FUNCTION_BLOCK SlitPairs
VAR_INPUT
	gap		:	AXIS_REF;
	centre	:	AXIS_REF;
	blade1	:	AXIS_REF;
	blade2	:	AXIS_REF;
	bCoupled	:	BOOL;
END_VAR
VAR_OUTPUT
END_VAR
VAR
	iState	:	UINT;
	MCCamInG	:	MC_CamIn_V2;
	MCCamInC	:	MC_CamIn_V2;
	MCCamAddG	:	MC_CamAdd;	
	MCCamAddC	:	MC_CamAdd;
	
	MCCamInB1	:	MC_CamIn_V2;
	MCCamInB2	:	MC_CamIn_V2;
	MCCamAddB1	:	MC_CamAdd;
	MCCamAddB2	:	MC_CamAdd;
	
	MCCamOutB1	:	MC_CamOut;
	MCCamOutB2	:	MC_CamOut;
	MCCamOutG	:	MC_CamOut;
	MCCamOutC	:	MC_CamOut;


	MCSetPosG	:	MC_SetPosition;
	MCSetPosC	:	MC_SetPosition;
	gapVal		:	LREAL;
	centVal		:	LREAL;
	

	
	
	
END_VAR

MCCamInB1(Master:=gap, Slave:=blade1);
MCCamAddB1(Master:=centre, Slave:=blade1);
MCCamInB2(Master:=gap, Slave:=blade2);
MCCamAddB2(Master:=centre, Slave:=blade2);

MCCamInG(Master:=blade1,Slave:=gap);
MCCamAddG(Master:=blade2, Slave:=gap);
MCCamInC(Master:=blade1, Slave:=centre);
MCCamAddC(Master:=blade2, Slave:=centre);

MCCamOutB1(Slave:=blade1);
MCCamOutB2(Slave:=blade2);
MCCamOutG(Slave:=gap);
MCCamOutC(Slave:=centre);


CASE iState OF
	0:	
		IF bCoupled THEN
			iState:=1;		//blades are slaves
		ELSE
			iState:= 30;		//blades are masters
		END_IF
	
	1:	//CAM IN THE GAP
		MCCamInB1(Master:=gap,Slave:=blade1,Execute:=TRUE,CamTableID:=1);
		MCCamInB2(Master:=gap,Slave:=blade2,Execute:=TRUE,CamTableID:=2);
		iState:=2;
	2:	//WAIT FOR CAM IN
		IF MCCamInB1.InSync AND MCCamInB2.InSync THEN
			MCCamInB1(Master:=gap,Slave:=blade1, Execute:=FALSE);
			MCCamInB2(Master:=gap,Slave:=blade2, Execute:=FALSE);
			iState:=3;
		END_IF
		
	3:	//CAM IN CENTRE
		MCCamAddB1(Master:=centre,Slave:=blade1,Execute:=TRUE,CamTableID:=3);
		MCCamAddB2(Master:=centre,Slave:=blade2,Execute:=TRUE,CamTableID:=4);
		iState:=4;
	4:	//WAIT FOR CAM IN
		IF MCCamAddB1.InSync AND MCCamAddB2.InSync THEN
			MCCamAddB1(Master:=centre,Slave:=blade1, Execute:=FALSE);
			MCCamAddB2(Master:=centre,Slave:=blade2, Execute:=FALSE);
			iState:=10;
		END_IF
	
	10:	//blades are slaves, do nothing unless this setup changes
		IF NOT bCoupled THEN
			iState:=20; //This is coming from slave blades, we now want to switch to gap and centre slaves so need to cam out first
		END_IF
		
	
		
	20:	//CAM OUT THE BLADES
		MCCamOutB1(Slave:=blade1, Execute:=TRUE);
		MCCamOutB2(Slave:=blade2, Execute:=TRUE);
		iState:=21;
	21:
		IF MCCamOutB1.Done AND MCCamOutB2.Done THEN
			MCCamOutB1(Slave:=blade1, Execute:=FALSE);
			MCCamOutB2(Slave:=blade2, Execute:=FALSE);
			iState:=30;	//CAMMED OUT READY FOR CAM IN
		END_IF

		
	30:	//CAM IN THE GAP AND CENTRES
		MCCamInG(Master:=blade1, Slave:=gap, Execute:=TRUE, CamTableID:= 5);
		MCCamInC(Master:=blade1, Slave:=centre, Execute:=TRUE, CamTableID:=6);
		iState:=31;
	
	31:
		IF MCCamInG.InSync AND MCCamInC.InSync THEN
			MCCamInG(Master:=blade1, Slave:=gap, Execute:=FALSE);
			MCCamInC(Master:=blade1, Slave:=centre, Execute:=FALSE);
			iState:=32;
		END_IF
	32:	//MULTI CAM
		MCCamAddG(Master:=blade2, Slave:=gap, Execute:=TRUE, CamTableID:=7);
		MCCamAddC(Master:=blade2, Slave:=centre, Execute:=TRUE, CamTableID:=8);
		iState:=33;
	33:
		IF MCCamAddG.InSync AND MCCamAddC.InSync THEN
			MCCamAddG(Master:=blade2, Slave:=gap, Execute:=FALSE);
			MCCamAddC(Master:=blade2, Slave:=centre, Execute:=FALSE);
			iState:=40;
		END_IF	
	
	40:	//blades are masters, do nothing unless changes
		IF bCoupled THEN
			iState:= 41;	//NEED TO CAM OUT
		END_IF
	41:
		MCCamOutG(Slave:=gap,Execute:=TRUE);
		MCCamOutC(Slave:=centre,Execute:=TRUE);
		iState:=42;
	42:
		IF MCCamOutG.Done AND MCCamOutC.Done THEN
			MCCamOutG(Slave:=gap, Execute:=FALSE);
			MCCamOutC(Slave:=centre, Execute:=FALSE);
			iState:=1;	//CAMMED OUT READY FOR CAM IN
		END_IF
		
END_CASE

END_FUNCTION_BLOCK

(* stored: Version 1.1.0.1, ProductVersion 3.1.4020.12
   POU SlitPairs: Id {c5204cda-557b-45d7-9676-d18cb5a98bfc}, SpecialFunc None *)
